// Mitsubishi GX Works2 project: fx3u cutup modbus   PLC: FX3U/FX3UC

PROGRAM MAIN
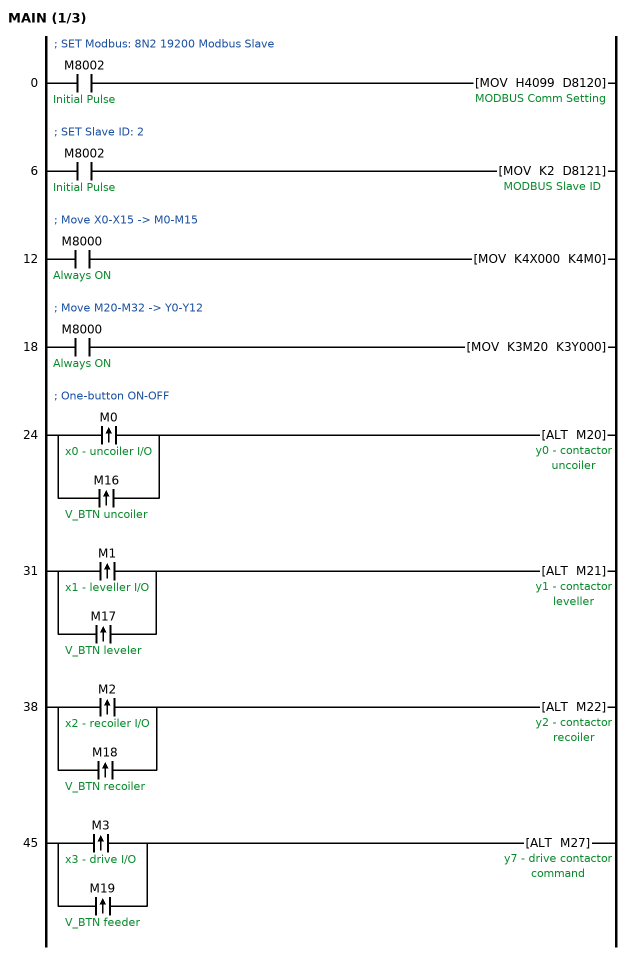
; SET Modbus: 8N2 19200 Modbus Slave
0     LD      M8002  ; Initial Pulse
      MOV     H4099 D8120  ; MODBUS Comm Setting
; SET Slave ID: 2
6     LD      M8002  ; Initial Pulse
      MOV     K2 D8121  ; MODBUS Slave ID
; Move X0-X15 -> M0-M15
12    LD      M8000  ; Always ON
      MOV     K4X000 K4M0  ; x0 - uncoiler I/O
; Move M20-M32 -> Y0-Y12
18    LD      M8000  ; Always ON
      MOV     K3M20 K3Y000  ; y0 - contactor uncoiler
; One-button ON-OFF
24    LDP     M0  ; x0 - uncoiler I/O
      ORP     M16  ; V_BTN uncoiler
      ALT     M20
31    LDP     M1  ; x1 - leveller I/O
      ORP     M17  ; V_BTN leveler
      ALT     M21  ; y1 - contactor leveller
38    LDP     M2  ; x2 - recoiler I/O
      ORP     M18  ; V_BTN recoiler
      ALT     M22  ; y2 - contactor recoiler
45    LDP     M3  ; x3 - drive I/O
      ORP     M19  ; V_BTN feeder
      ALT     M27  ; y7 - drive contactor command
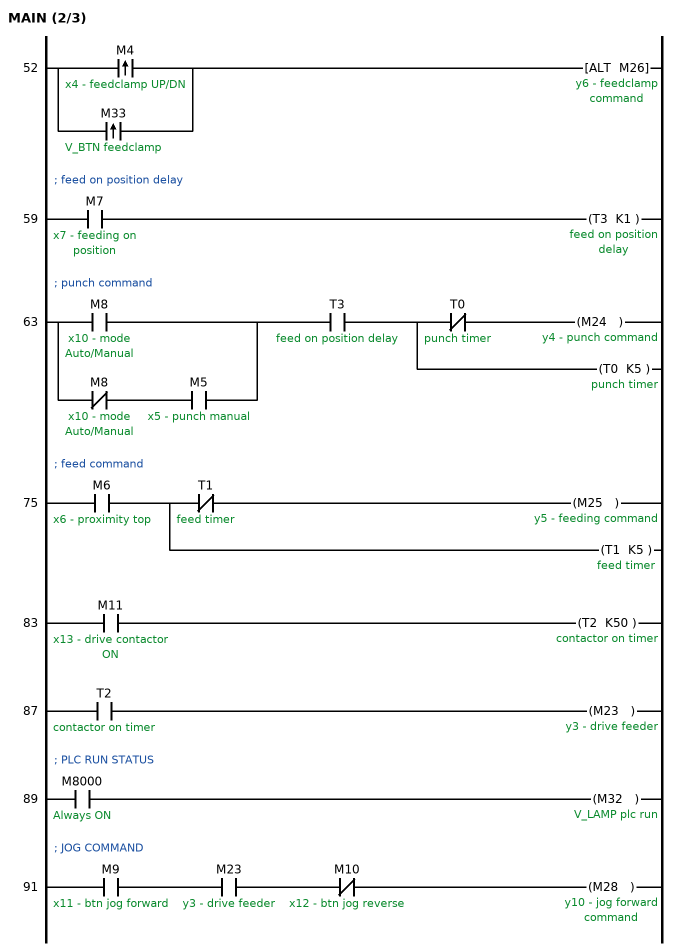
52    LDP     M4  ; x4 - feedclamp UP/DN
      ORP     M33  ; V_BTN feedclamp
      ALT     M26  ; y6 - feedclamp command
; feed on position delay
59    LD      M7  ; x7 - feeding on position
      OUT     T3 K1  ; feed on position delay
; punch command
63    LD      M8  ; x10 - mode Auto/Manual
      LDI     M8  ; x10 - mode Auto/Manual
      AND     M5  ; x5 - punch manual
      ORB
      AND     T3  ; feed on position delay
      MPS
      ANI     T0  ; punch timer
      OUT     M24  ; y4 - punch command
      MPP
      OUT     T0 K5  ; punch timer
; feed command
75    LD      M6  ; x6 - proximity top
      MPS
      ANI     T1  ; feed timer
      OUT     M25  ; y5 - feeding command
      MPP
      OUT     T1 K5  ; feed timer
83    LD      M11  ; x13 - drive contactor ON
      OUT     T2 K50  ; contactor on timer
87    LD      T2  ; contactor on timer
      OUT     M23  ; y3 - drive feeder
; PLC RUN STATUS
89    LD      M8000  ; Always ON
      OUT     M32  ; V_LAMP plc run
; JOG COMMAND
91    LD      M9  ; x11 - btn jog forward
      AND     M23  ; y3 - drive feeder
      ANI     M10  ; x12 - btn jog reverse
      OUT     M28  ; y10 - jog forward command
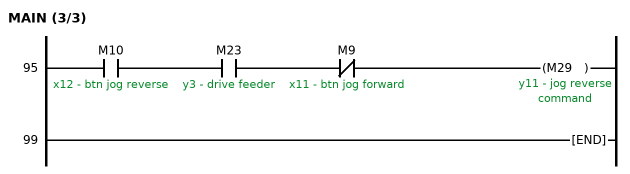
95    LD      M10  ; x12 - btn jog reverse
      AND     M23  ; y3 - drive feeder
      ANI     M9  ; x11 - btn jog forward
      OUT     M29  ; y11 - jog reverse command
99    END
END_PROGRAM

// device comments not shown above
M15  ; ##RESERVED##
M12  ; x14
M13  ; x15
